TYPE CmpConvBreakStopGroupConfig :
STRUCT
	NumberStops: DINT;
	BreakStopDefault: BreakStopConfig;
	BreakStops: ARRAY[1..cBreakStopGroupMaxInstance] OF BreakStopConfig;
END_STRUCT
END_TYPE

(* stored: Version 1.1.0.1, ProductVersion 3.1.4024.6
   DUT CmpConvBreakStopGroupConfig: Id {336b3df1-683c-4d1f-865a-aee7a0a17094} *)
